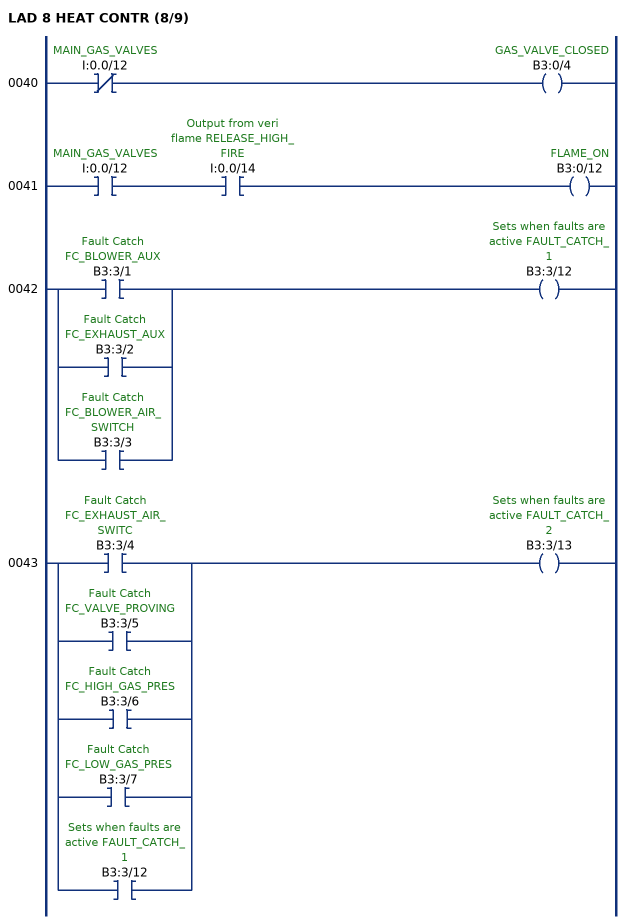
% Rung: 40 %
SOR XIO I:0.0/12 OTE B3:0/4 EOR
%   I:0.0/12  MAIN_GAS_VALVES %
%   B3:0/4  GAS_VALVE_CLOSED %
% Rung: 41 %
SOR XIC I:0.0/12 XIC I:0.0/14 OTE B3:0/12 EOR
%   I:0.0/12  MAIN_GAS_VALVES %
%   I:0.0/14  RELEASE_HIGH_FIRE  "Output from veri flame" %
%   B3:0/12  FLAME_ON %
% Rung: 42 %
SOR BST XIC B3:3/1 NXB BST XIC B3:3/2 NXB XIC B3:3/3 BND BND OTE B3:3/12 EOR
%   B3:3/1  FC_BLOWER_AUX  "Fault Catch" %
%   B3:3/2  FC_EXHAUST_AUX  "Fault Catch" %
%   B3:3/3  FC_BLOWER_AIR_SWITCH  "Fault Catch" %
%   B3:3/12  FAULT_CATCH_1  "Sets when faults are active" %
% Rung: 43 %
SOR BST XIC B3:3/4 NXB BST XIC B3:3/5 NXB BST XIC B3:3/6 NXB BST XIC B3:3/7 NXB XIC B3:3/12 BND BND BND BND OTE B3:3/13 EOR
%   B3:3/4  FC_EXHAUST_AIR_SWITC  "Fault Catch" %
%   B3:3/5  FC_VALVE_PROVING  "Fault Catch" %
%   B3:3/6  FC_HIGH_GAS_PRES  "Fault Catch" %
%   B3:3/7  FC_LOW_GAS_PRES  "Fault Catch" %
%   B3:3/12  FAULT_CATCH_1  "Sets when faults are active" %
%   B3:3/13  FAULT_CATCH_2  "Sets when faults are active" %

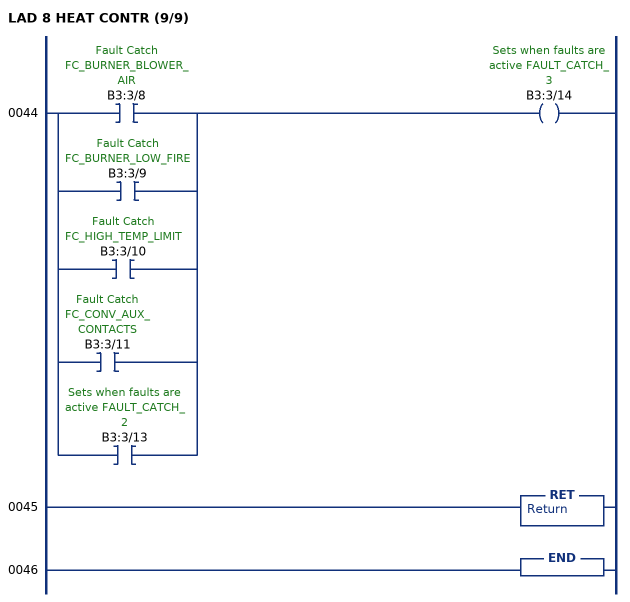
% Rung: 44 %
SOR BST XIC B3:3/8 NXB BST XIC B3:3/9 NXB BST XIC B3:3/10 NXB BST XIC B3:3/11 NXB XIC B3:3/13 BND BND BND BND OTE B3:3/14 EOR
%   B3:3/8  FC_BURNER_BLOWER_AIR  "Fault Catch" %
%   B3:3/9  FC_BURNER_LOW_FIRE  "Fault Catch" %
%   B3:3/10  FC_HIGH_TEMP_LIMIT  "Fault Catch" %
%   B3:3/11  FC_CONV_AUX_CONTACTS  "Fault Catch" %
%   B3:3/13  FAULT_CATCH_2  "Sets when faults are active" %
%   B3:3/14  FAULT_CATCH_3  "Sets when faults are active" %
% Rung: 45 %
SOR RET EOR
% Rung: 46 %
SOR END EOR

LADDER 9 "CLR FAULTS"
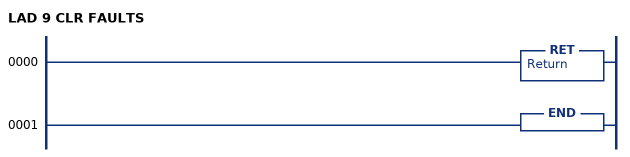
% Rung: 0 %
SOR RET EOR
% Rung: 1 %
SOR END EOR

LADDER 10 "HOUR METER"
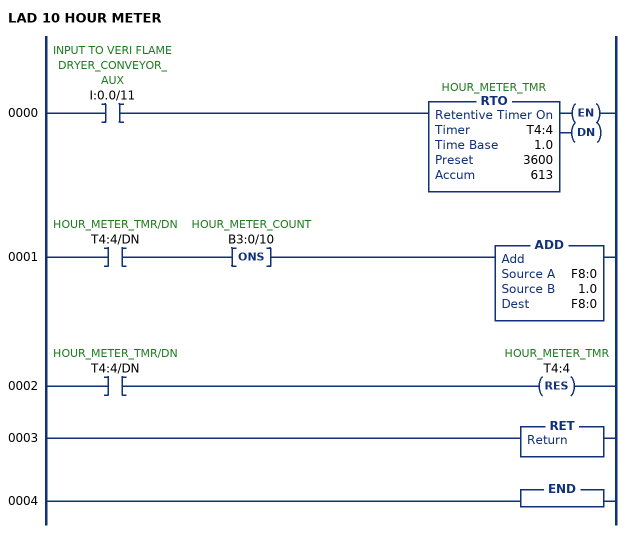
% Rung: 0 %
SOR XIC I:0.0/11 RTO T4:4 1.0 3600 613 EOR
%   I:0.0/11  DRYER_CONVEYOR_AUX  "INPUT TO VERI FLAME" %
%   T4:4  HOUR_METER_TMR %
% Rung: 1 %
SOR XIC T4:4/DN ONS B3:0/10 ADD F8:0 1.0 F8:0 EOR
%   T4:4  HOUR_METER_TMR %
%   B3:0/10  HOUR_METER_COUNT %
% Rung: 2 %
SOR XIC T4:4/DN RES T4:4 EOR
%   T4:4  HOUR_METER_TMR %
% Rung: 3 %
SOR RET EOR
% Rung: 4 %
SOR END EOR

LADDER 11 "CONV CLEAN"
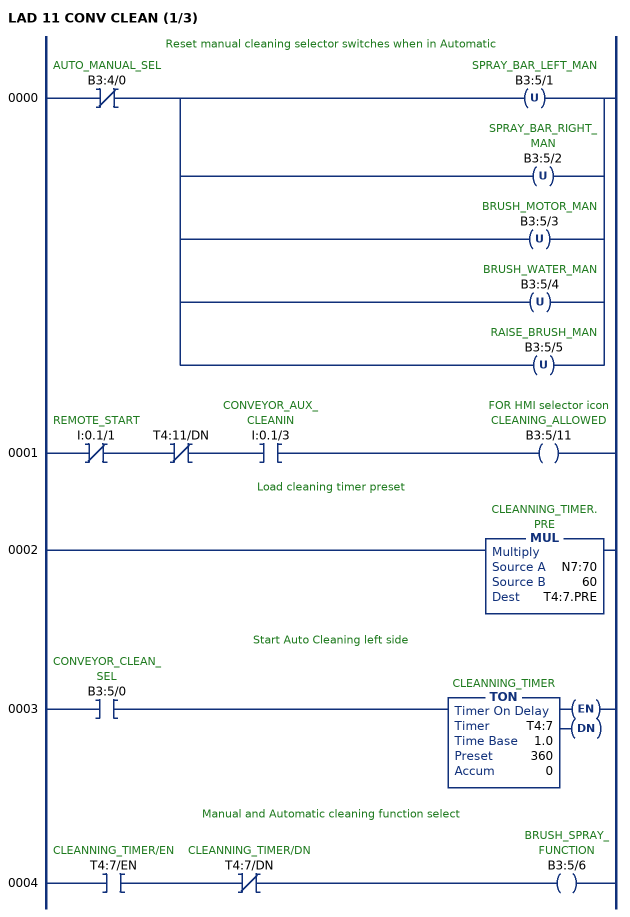
% Rung: 0 %
% Reset manual cleaning selector switches when in Automatic %
SOR XIO B3:4/0 BST OTU B3:5/1 NXB BST OTU B3:5/2 NXB BST OTU B3:5/3 NXB BST OTU B3:5/4 NXB OTU B3:5/5 BND BND BND BND EOR
%   B3:4/0  AUTO_MANUAL_SEL %
%   B3:5/1  SPRAY_BAR_LEFT_MAN %
%   B3:5/2  SPRAY_BAR_RIGHT_MAN %
%   B3:5/3  BRUSH_MOTOR_MAN %
%   B3:5/4  BRUSH_WATER_MAN %
%   B3:5/5  RAISE_BRUSH_MAN %
% Rung: 1 %
SOR XIO I:0.1/1 XIO T4:11/DN XIC I:0.1/3 OTE B3:5/11 EOR
%   I:0.1/1  REMOTE_START %
%   I:0.1/3  CONVEYOR_AUX_CLEANIN %
%   B3:5/11  CLEANING_ALLOWED  "FOR HMI selector icon" %
% Rung: 2 %
% Load cleaning timer preset %
SOR MUL N7:70 60 T4:7.PRE EOR
%   N7:70  CLEANING_TIME %
%   T4:7  CLEANNING_TIMER %
% Rung: 3 %
% Start Auto Cleaning left side %
SOR XIC B3:5/0 TON T4:7 1.0 360 0 EOR
%   B3:5/0  CONVEYOR_CLEAN_SEL %
%   T4:7  CLEANNING_TIMER %
% Rung: 4 %
% Manual and Automatic cleaning function select %
SOR XIC T4:7/EN XIO T4:7/DN OTE B3:5/6 EOR
%   T4:7  CLEANNING_TIMER %
%   B3:5/6  BRUSH_SPRAY_FUNCTION %

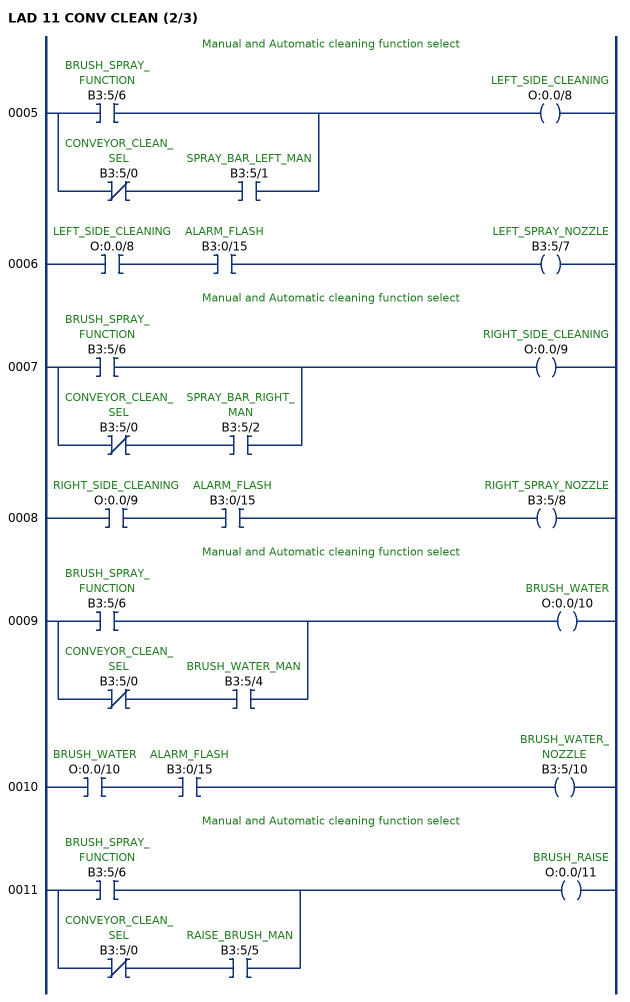
% Rung: 5 %
% Manual and Automatic cleaning function select %
SOR BST XIC B3:5/6 NXB XIO B3:5/0 XIC B3:5/1 BND OTE O:0.0/8 EOR
%   B3:5/6  BRUSH_SPRAY_FUNCTION %
%   B3:5/0  CONVEYOR_CLEAN_SEL %
%   B3:5/1  SPRAY_BAR_LEFT_MAN %
%   O:0.0/8  LEFT_SIDE_CLEANING %
% Rung: 6 %
SOR XIC O:0.0/8 XIC B3:0/15 OTE B3:5/7 EOR
%   O:0.0/8  LEFT_SIDE_CLEANING %
%   B3:0/15  ALARM_FLASH %
%   B3:5/7  LEFT_SPRAY_NOZZLE %
% Rung: 7 %
% Manual and Automatic cleaning function select %
SOR BST XIC B3:5/6 NXB XIO B3:5/0 XIC B3:5/2 BND OTE O:0.0/9 EOR
%   B3:5/6  BRUSH_SPRAY_FUNCTION %
%   B3:5/0  CONVEYOR_CLEAN_SEL %
%   B3:5/2  SPRAY_BAR_RIGHT_MAN %
%   O:0.0/9  RIGHT_SIDE_CLEANING %
% Rung: 8 %
SOR XIC O:0.0/9 XIC B3:0/15 OTE B3:5/8 EOR
%   O:0.0/9  RIGHT_SIDE_CLEANING %
%   B3:0/15  ALARM_FLASH %
%   B3:5/8  RIGHT_SPRAY_NOZZLE %
% Rung: 9 %
% Manual and Automatic cleaning function select %
SOR BST XIC B3:5/6 NXB XIO B3:5/0 XIC B3:5/4 BND OTE O:0.0/10 EOR
%   B3:5/6  BRUSH_SPRAY_FUNCTION %
%   B3:5/0  CONVEYOR_CLEAN_SEL %
%   B3:5/4  BRUSH_WATER_MAN %
%   O:0.0/10  BRUSH_WATER %
% Rung: 10 %
SOR XIC O:0.0/10 XIC B3:0/15 OTE B3:5/10 EOR
%   O:0.0/10  BRUSH_WATER %
%   B3:0/15  ALARM_FLASH %
%   B3:5/10  BRUSH_WATER_NOZZLE %
% Rung: 11 %
% Manual and Automatic cleaning function select %
SOR BST XIC B3:5/6 NXB XIO B3:5/0 XIC B3:5/5 BND OTE O:0.0/11 EOR
%   B3:5/6  BRUSH_SPRAY_FUNCTION %
%   B3:5/0  CONVEYOR_CLEAN_SEL %
%   B3:5/5  RAISE_BRUSH_MAN %
%   O:0.0/11  BRUSH_RAISE %

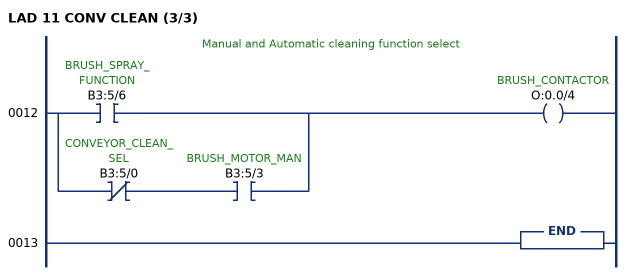
% Rung: 12 %
% Manual and Automatic cleaning function select %
SOR BST XIC B3:5/6 NXB XIO B3:5/0 XIC B3:5/3 BND OTE O:0.0/4 EOR
%   B3:5/6  BRUSH_SPRAY_FUNCTION %
%   B3:5/0  CONVEYOR_CLEAN_SEL %
%   B3:5/3  BRUSH_MOTOR_MAN %
%   O:0.0/4  BRUSH_CONTACTOR %
% Rung: 13 %
SOR END EOR

OTHER DOCUMENTED ADDRESSES
  B3:0/11  FLAME_STANDBY
  B3:0/14  SET_MIN_VFD_SPEED
  B3:4/6  DISPLAY_CONVEYOR_DEL
  B3:10/0  "Lube Run Enable request from CLX 1 Write message"
  I:0.1/0  VALVE_PROVING_ALARM
  I:0.1/2  DN_STREAM_CONV_AUX
  I:1.0/0  TC1
  I:2.0/0  SENSOR_PLENUM
  I:2.0/1  SENSOR_RETURN
  I:2.1/0  SENSOR_Q
  I:2.2/0  SENSOR_HUMIDITY
  I:2.3/0  SENSOR_TEMP_RHL
  N7:23  HUMIDITY_SCALING_MUL  "Value needed to scale output"
  N7:25  HUMITITY_MIN_SETPOIN
  N7:30  TEMP_RHL_SENSOR  "RH Sensor Temperature"
  N7:32  SCALE_TEMPERATUR_DIV  "Value needed to adjust output to degrees fahrenheit"
  N7:46  PLENUM_PS_ALARM
  PD9:0.3  "SPS Setpoint"
  PFILE:5  "a"
  Q4:1  END_OF_VALVE_POS
  RST  
  SET  "s:5/0"

COMMENTS NOT ATTACHED TO A CURRENT RUNG
  N7:3: Subract to bring sensor value to zero
  N7:53: Find slope intercept  b value step #2 -  multiply point Ax times slope
  N7:50: Find slope step #2 -  multiply Y dif by 100 to get better accuracy
  N7:56: Solve for speed Step #2 - divide by 100 (multiply slope times humidity)
  N7:55: Find slope intercept  b value step #5 -  sub Ay minus Ax*slope
  N7:54: Find slope intercept  b value step #3 -  multiply point Ay by 100 for Accuracy
  N7:63: Calculates the temperature difference on start up to open the fan butterfly valve fully to build heat faster when cold.

DATA TABLE (non-zero values as saved)
DATA B3
% B3:0 % 0X0000 0X8000 0X0000 0X0000 0X0180 0X0000 0X0000 0X0100 0X0000 0X0000
% B3:10 % 0X0001 0X0000 0X0000 0X0000 0X0000 0X0000 0X0000 0X0000 0X0000 0X0000
DATA T4
% .PRE .ACC %
% T4:0 % 299 0
% T4:1 % 1 0
% T4:2 % 150 0
% T4:3 % 100 0
% T4:4 % 3600 613
% T4:5 % 45 45
% T4:6 % 4 0
% T4:7 % 360 0
% T4:8 % 600 0
% T4:9 % 1800 0
% T4:10 % 9999 0
% T4:11 % 30 30
% T4:12 % 30 20
DATA N7
% N7:0 % 6956 6226 105 1 7 6280 6265 18 1 1
% N7:10 % 450 448 451 1349 300 1650 1350 1349 11572 3400
% N7:20 % 8968 6250 240 10 26 25 5 60 100 12
% N7:30 % 10 0 195 11076 16277 5 299 135 3 30
% N7:40 % 2 1 3 200 1200 5 0 0 0 1350
% N7:50 % 85 10 0 0 60 1 20 20 0 0
% N7:60 % 45 0 0 0 0 0 0 0 0 0
% N7:70 % 6 0 0 0 0 0 0
DATA F8
% F8:0 % 14
